FUNCTION_BLOCK VFD IMPLEMENTS itfAutoManual
VAR_INPUT
	VFDInput : VFDI;
END_VAR
VAR_OUTPUT
	VFDOutput : VFDO;
END_VAR
VAR
	MotorComp : Motor;
	MotorIref : REFERENCE TO MotorI;
	MotorOref : REFERENCE TO MotorO;

	ScaleComp : itfScaleAnalogOutputImplement;
	Scale : itfScale;

	RampComp : itfRampImplement;
	Ramp : itfRamp;
	
	CoilR : R_TRIG;
	CoilF : F_TRIG;
	
	FlagUp : BOOL;
	FlagDown : BOOL;
END_VAR

Map();

CoilR(CLK:= MotorOref.Coil);
CoilF(CLK:= MotorOref.Coil);

METHOD PRIVATE Map : BOOL
VAR_INPUT
END_VAR
MotorIref REF= VFDInput;
MotorOref REF= VFDOutput;
MotorComp(MotorInput := MotorIref, MotorOutput => MotorOref);

Scale := ScaleComp;
Ramp := RampComp;

Ramp.pTargetFreq := VFDInput.InputFreq;
Ramp.pRampRate := VFDInput.RampRate;

Scale.pMaxSignalValue := VFDInput.FreqMaxSignal;
Scale.pAnalogSignal := Ramp.pOutputValue;
VFDOutput.OutputFreq := Scale.pScaledSignal;
Scale.mScale();
END_METHOD

{warning 'add method implementation '}
METHOD mAutoOff : BOOL
RampFreq();
MotorComp.mAutoOff();
END_METHOD

{warning 'add method implementation '}
METHOD mAutoOn : BOOL
RampFreq();
MotorComp.mAutoOn();
END_METHOD

{warning 'add method implementation '}
METHOD mFault : BOOL
mFault := MotorComp.mFault();
END_METHOD

{warning 'add method implementation '}
METHOD mManual : BOOL
RampFreq();
MotorComp.mManual();
END_METHOD

{warning 'add method implementation '}
METHOD mRunning : BOOL
mRunning := MotorComp.mRunning();
END_METHOD

METHOD RampFreq : INT
VAR_INPUT
END_VAR
IF CoilR.Q THEN
	FlagUp := TRUE;
	// Setting Flag
	FlagDown := FALSE;
END_IF

IF CoilF.Q THEN
	FlagDown := TRUE;
	// Setting Flag
	FlagUp := FALSE;
END_IF

IF FlagUp THEN
	//FlagDown := FALSE;
	Ramp.mRampUp();
	IF Ramp.pRampDone THEN
		FlagUp := FALSE;
	END_IF
END_IF

IF FlagDown THEN
	//FlagUp := FALSE;
	Ramp.mRampDown();
	IF Ramp.pOutputValue = 0 THEN
		FlagDown := FALSE;
	END_IF
END_IF
END_METHOD

END_FUNCTION_BLOCK

(* stored: Version 1.1.0.1, ProductVersion 3.1.4024.12
   POU VFD: Id {65cf7e09-36be-4f79-ada8-7d2f724d4ada}, SpecialFunc None
   Method Map: Id {6f960a0f-f7ad-4b89-9aeb-006fd4128c60}
   Method mAutoOff: Id {996be5e1-25a8-4124-8af7-e5c0e98b76f7}
   Method mAutoOn: Id {e1420c6f-48e5-4cc2-9621-24907e96929e}
   Method mFault: Id {c06fde52-78da-4c8a-b4af-4b11cb752da9}
   Method mManual: Id {d480ba3f-794a-4551-a7fa-cbf86b384f97}
   Method mRunning: Id {34b66f92-d3a1-4b1d-a570-870cc696ecca}
   Method RampFreq: Id {32df45e3-b7b0-4700-a55a-f26e3803b2b7} *)
